{attribute 'no_check'}
//Overwrite function - Returns velocity setpoint based on max velo and requested overwrite 
FUNCTION getOvrVelo : LREAL
VAR_INPUT
	SetVelo													:	LREAL;
	MaxVelo													:	LREAL;
END_VAR
VAR
END_VAR

IF 	MaxVelo = 0.0 OR SetVelo = 0.0
THEN
	GetOvrVelo 												:= 0.0;
ELSE                										
	GetOvrVelo 												:= 100.0 / MaxVelo * SetVelo;
END_IF

END_FUNCTION

(* stored: Version 1.1.0.1, ProductVersion 3.1.4024.3
   POU getOvrVelo: Id {fdae079d-c334-47c4-bf89-4e30fa852178}, SpecialFunc None *)
